FUNCTION_BLOCK EL_NeedleAxis (* NeedleAxis logic: command -> outputs (break before make), inputs -> state channel *)
  (* Standard: 61499-2 *)
  (* Version 0.1, 2026-09-28, Project contributors, AAU Smart Production Lab *)
  PACKAGE filler;
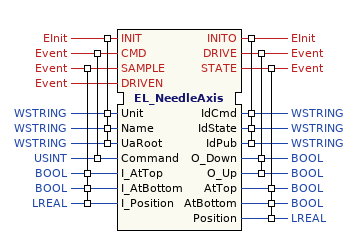
  EVENT_INPUT
    INIT : EInit WITH Unit, Name, UaRoot;
    CMD WITH Command;
    SAMPLE WITH I_AtTop, I_AtBottom, I_Position;
    DRIVEN;
  END_EVENT
  EVENT_OUTPUT
    INITO : EInit WITH IdCmd, IdState, IdPub;
    DRIVE WITH O_Down, O_Up;
    STATE WITH AtTop, AtBottom, Position;
  END_EVENT
  VAR_INPUT
    Unit : WSTRING;
    Name : WSTRING;
    UaRoot : WSTRING;
    Command : USINT;
    I_AtTop : BOOL;
    I_AtBottom : BOOL;
    I_Position : LREAL;
  END_VAR
  VAR_OUTPUT
    IdCmd : WSTRING;
    IdState : WSTRING;
    IdPub : WSTRING;
    O_Down : BOOL;
    O_Up : BOOL;
    AtTop : BOOL;
    AtBottom : BOOL;
    Position : LREAL;
  END_VAR
  VAR
    N_Down : BOOL;
    N_Up : BOOL;
  END_VAR
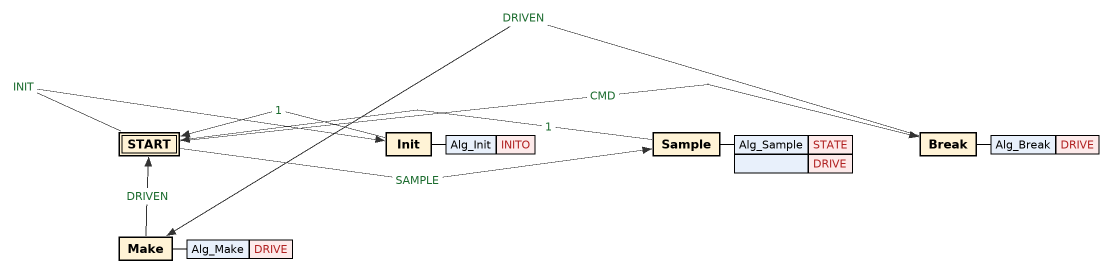
  EC_STATES
    START;
    Init : Alg_Init -> INITO;
    Sample : Alg_Sample -> STATE, -> DRIVE;
    Break : Alg_Break -> DRIVE;
    Make : Alg_Make -> DRIVE;
  END_STATES
  EC_TRANSITIONS
    START TO Init := INIT;
    START TO Sample := SAMPLE;
    START TO Break := CMD;
    Init TO START := 1;
    Sample TO START := 1;
    Break TO Make := DRIVEN;
    Make TO START := DRIVEN;
  END_TRANSITIONS
  ALGORITHM Alg_Init IN ST:
IdCmd := CONCAT(CONCAT(CONCAT(CONCAT("loc[", Unit), "/"), Name), "/cmd]");
IdState := CONCAT(CONCAT(CONCAT(CONCAT("loc[", Unit), "/"), Name), "/state]");
IdPub := CONCAT(CONCAT(CONCAT(CONCAT(CONCAT(CONCAT(CONCAT(CONCAT(CONCAT(CONCAT(CONCAT(CONCAT("opc_ua[WRITE;", UaRoot), "/Equipment/"), Name), "/AtTop;"), UaRoot), "/Equipment/"), Name), "/AtBottom;"), UaRoot), "/Equipment/"), Name), "/Position]");
  END_ALGORITHM
  ALGORITHM Alg_Sample IN ST:
AtTop := I_AtTop;
AtBottom := I_AtBottom;
Position := I_Position;
  END_ALGORITHM
  ALGORITHM Alg_Break IN ST:
N_Down := (Command = 1);
N_Up := (Command = 2);
O_Down := O_Down AND N_Down;
O_Up := O_Up AND N_Up;
  END_ALGORITHM
  ALGORITHM Alg_Make IN ST:
N_Down := (Command = 1);
N_Up := (Command = 2);
O_Down := N_Down;
O_Up := N_Up;
  END_ALGORITHM
END_FUNCTION_BLOCK
